FUNCTION_BLOCK TM_DI32 (* Composite Function Block Type *)
  (* Standard: 61499-2 *)
  (* Version 0.0, 18/08/2026, template *)
  PACKAGE Hidryco.HidrycoLib;
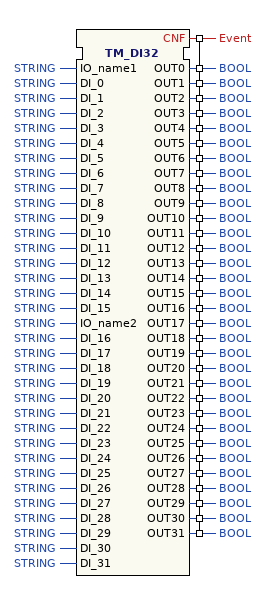
  EVENT_OUTPUT
    CNF WITH OUT0, OUT1, OUT2, OUT3, OUT4, OUT5, OUT6, OUT7, OUT8, OUT9, OUT10, OUT11, OUT12, OUT13, OUT14, OUT15, OUT16, OUT17, OUT18, OUT19, OUT20, OUT21, OUT22, OUT23, OUT24, OUT25, OUT26, OUT27, OUT28, OUT29, OUT30, OUT31;
  END_EVENT
  VAR_INPUT
    IO_name1 : STRING;
    DI_0 : STRING;
    DI_1 : STRING;
    DI_2 : STRING;
    DI_3 : STRING;
    DI_4 : STRING;
    DI_5 : STRING;
    DI_6 : STRING;
    DI_7 : STRING;
    DI_8 : STRING;
    DI_9 : STRING;
    DI_10 : STRING;
    DI_11 : STRING;
    DI_12 : STRING;
    DI_13 : STRING;
    DI_14 : STRING;
    DI_15 : STRING;
    IO_name2 : STRING;
    DI_16 : STRING;
    DI_17 : STRING;
    DI_18 : STRING;
    DI_19 : STRING;
    DI_20 : STRING;
    DI_21 : STRING;
    DI_22 : STRING;
    DI_23 : STRING;
    DI_24 : STRING;
    DI_25 : STRING;
    DI_26 : STRING;
    DI_27 : STRING;
    DI_28 : STRING;
    DI_29 : STRING;
    DI_30 : STRING;
    DI_31 : STRING;
  END_VAR
  VAR_OUTPUT
    OUT0 : BOOL; (* Output bit image, bit 0 is the LSB of OUT1 *)
    OUT1 : BOOL; (* Output bit image, bit 0 is the LSB of OUT1 *)
    OUT2 : BOOL; (* Output bit image, bit 0 is the LSB of OUT1 *)
    OUT3 : BOOL; (* Output bit image, bit 0 is the LSB of OUT1 *)
    OUT4 : BOOL; (* Output bit image, bit 0 is the LSB of OUT1 *)
    OUT5 : BOOL; (* Output bit image, bit 0 is the LSB of OUT1 *)
    OUT6 : BOOL; (* Output bit image, bit 0 is the LSB of OUT1 *)
    OUT7 : BOOL; (* Output bit image, bit 0 is the LSB of OUT1 *)
    OUT8 : BOOL; (* Output bit image, bit 0 is the LSB of OUT1 *)
    OUT9 : BOOL; (* Output bit image, bit 0 is the LSB of OUT1 *)
    OUT10 : BOOL; (* Output bit image, bit 0 is the LSB of OUT1 *)
    OUT11 : BOOL; (* Output bit image, bit 0 is the LSB of OUT1 *)
    OUT12 : BOOL; (* Output bit image, bit 0 is the LSB of OUT1 *)
    OUT13 : BOOL; (* Output bit image, bit 0 is the LSB of OUT1 *)
    OUT14 : BOOL; (* Output bit image, bit 0 is the LSB of OUT1 *)
    OUT15 : BOOL; (* Output bit image, bit 0 is the LSB of OUT1 *)
    OUT16 : BOOL; (* Output bit image, bit 0 is the LSB of OUT1 *)
    OUT17 : BOOL; (* Output bit image, bit 0 is the LSB of OUT1 *)
    OUT18 : BOOL; (* Output bit image, bit 0 is the LSB of OUT1 *)
    OUT19 : BOOL; (* Output bit image, bit 0 is the LSB of OUT1 *)
    OUT20 : BOOL; (* Output bit image, bit 0 is the LSB of OUT1 *)
    OUT21 : BOOL; (* Output bit image, bit 0 is the LSB of OUT1 *)
    OUT22 : BOOL; (* Output bit image, bit 0 is the LSB of OUT1 *)
    OUT23 : BOOL; (* Output bit image, bit 0 is the LSB of OUT1 *)
    OUT24 : BOOL; (* Output bit image, bit 0 is the LSB of OUT1 *)
    OUT25 : BOOL; (* Output bit image, bit 0 is the LSB of OUT1 *)
    OUT26 : BOOL; (* Output bit image, bit 0 is the LSB of OUT1 *)
    OUT27 : BOOL; (* Output bit image, bit 0 is the LSB of OUT1 *)
    OUT28 : BOOL; (* Output bit image, bit 0 is the LSB of OUT1 *)
    OUT29 : BOOL; (* Output bit image, bit 0 is the LSB of OUT1 *)
    OUT30 : BOOL; (* Output bit image, bit 0 is the LSB of OUT1 *)
    OUT31 : BOOL; (* Output bit image, bit 0 is the LSB of OUT1 *)
  END_VAR
  FBS
    BITMAN1 : BITMAN_1879143E4E6E9A030; {SET_ATTRIBUTE(Configuration.GenericFBType.InterfaceParams, Runtime.Standard#CNTIN:=1;CNTOUT:=16;IN${CNTIN$}:WORD;OUT${CNTOUT$}:BOOL,BOOL,BOOL,BOOL,BOOL,BOOL,BOOL,BOOL,BOOL,BOOL,BOOL,BOOL,BOOL,BOOL,BOOL,BOOL)}
    SYMLINKMULTIVARDST3 : SYMLINKMULTIVARDST_5A03F112CD5D470(QI := TRUE); {SET_ATTRIBUTE(Configuration.GenericFBType.InterfaceParams, Runtime.System#I:=1;VALUE${I$}:INT)}
    ANY2ANY1 : ANY2ANY_100577755E31233DE; {SET_ATTRIBUTE(Configuration.GenericFBType.InterfaceParams, Runtime.Standard#CNT:=1;IN${CNT$}:INT;OUT${CNT$}:WORD)}
    TM : SYMLINKMULTIVARSRC_854A896E88500D19(QI := TRUE); {SET_ATTRIBUTE(Configuration.GenericFBType.InterfaceParams, Runtime.System#I:=16;VALUE${I$}:BOOL,BOOL,BOOL,BOOL,BOOL,BOOL,BOOL,BOOL,BOOL,BOOL,BOOL,BOOL,BOOL,BOOL,BOOL,BOOL)}
    plcStart1 : plcStart(Prio := 3);
    BITMAN2 : BITMAN_1879143E4E6E9A030; {SET_ATTRIBUTE(Configuration.GenericFBType.InterfaceParams, Runtime.Standard#CNTIN:=1;CNTOUT:=16;IN${CNTIN$}:WORD;OUT${CNTOUT$}:BOOL,BOOL,BOOL,BOOL,BOOL,BOOL,BOOL,BOOL,BOOL,BOOL,BOOL,BOOL,BOOL,BOOL,BOOL,BOOL)}
    SYMLINKMULTIVARDST4 : SYMLINKMULTIVARDST_5A03F112CD5D470(QI := TRUE); {SET_ATTRIBUTE(Configuration.GenericFBType.InterfaceParams, Runtime.System#I:=1;VALUE${I$}:INT)}
    ANY2ANY2 : ANY2ANY_100577755E31233DE; {SET_ATTRIBUTE(Configuration.GenericFBType.InterfaceParams, Runtime.Standard#CNT:=1;IN${CNT$}:INT;OUT${CNT$}:WORD)}
    TM1 : SYMLINKMULTIVARSRC_854A896E88500D19(QI := TRUE); {SET_ATTRIBUTE(Configuration.GenericFBType.InterfaceParams, Runtime.System#I:=16;VALUE${I$}:BOOL,BOOL,BOOL,BOOL,BOOL,BOOL,BOOL,BOOL,BOOL,BOOL,BOOL,BOOL,BOOL,BOOL,BOOL,BOOL)}
    plcStart2 : plcStart(Prio := 3);
    FB1 : E_MERGE;
  END_FBS
  EVENT_CONNECTIONS
    SYMLINKMULTIVARDST3.CNF TO ANY2ANY1.REQ;
    ANY2ANY1.CNF TO BITMAN1.REQ;
    SYMLINKMULTIVARDST3.INITO TO BITMAN1.INIT;
    BITMAN1.INITO TO TM.INIT;
    BITMAN1.CNF TO TM.REQ;
    plcStart1.FIRST_INIT TO SYMLINKMULTIVARDST3.INIT;
    plcStart1.REDO_INIT TO SYMLINKMULTIVARDST3.INIT;
    TM.INITO TO plcStart1.ACK_FIRST;
    SYMLINKMULTIVARDST4.CNF TO ANY2ANY2.REQ;
    ANY2ANY2.CNF TO BITMAN2.REQ;
    SYMLINKMULTIVARDST4.INITO TO BITMAN2.INIT;
    BITMAN2.INITO TO TM1.INIT;
    BITMAN2.CNF TO TM1.REQ;
    plcStart2.FIRST_INIT TO SYMLINKMULTIVARDST4.INIT;
    plcStart2.REDO_INIT TO SYMLINKMULTIVARDST4.INIT;
    TM1.INITO TO plcStart2.ACK_FIRST;
    BITMAN2.CNF TO FB1.EI2;
    BITMAN1.CNF TO FB1.EI1;
    FB1.EO TO CNF;
  END_CONNECTIONS
  DATA_CONNECTIONS
    SYMLINKMULTIVARDST3.VALUE1 TO ANY2ANY1.IN1;
    ANY2ANY1.OUT1 TO BITMAN1.IN1;
    BITMAN1.OUT1 TO TM.VALUE1;
    BITMAN1.OUT2 TO TM.VALUE2;
    BITMAN1.OUT3 TO TM.VALUE3;
    BITMAN1.OUT4 TO TM.VALUE4;
    BITMAN1.OUT5 TO TM.VALUE5;
    BITMAN1.OUT6 TO TM.VALUE6;
    BITMAN1.OUT7 TO TM.VALUE7;
    BITMAN1.OUT8 TO TM.VALUE8;
    BITMAN1.OUT9 TO TM.VALUE9;
    BITMAN1.OUT10 TO TM.VALUE10;
    BITMAN1.OUT11 TO TM.VALUE11;
    BITMAN1.OUT12 TO TM.VALUE12;
    BITMAN1.OUT13 TO TM.VALUE13;
    BITMAN1.OUT14 TO TM.VALUE14;
    BITMAN1.OUT15 TO TM.VALUE15;
    BITMAN1.OUT16 TO TM.VALUE16;
    IO_name1 TO SYMLINKMULTIVARDST3.NAME1;
    DI_0 TO TM.NAME1;
    DI_1 TO TM.NAME2;
    DI_2 TO TM.NAME3;
    DI_3 TO TM.NAME4;
    DI_4 TO TM.NAME5;
    DI_5 TO TM.NAME6;
    DI_6 TO TM.NAME7;
    DI_7 TO TM.NAME8;
    DI_8 TO TM.NAME9;
    DI_9 TO TM.NAME10;
    DI_10 TO TM.NAME11;
    DI_11 TO TM.NAME12;
    DI_12 TO TM.NAME13;
    DI_13 TO TM.NAME14;
    DI_14 TO TM.NAME15;
    DI_15 TO TM.NAME16;
    SYMLINKMULTIVARDST4.VALUE1 TO ANY2ANY2.IN1;
    ANY2ANY2.OUT1 TO BITMAN2.IN1;
    BITMAN2.OUT1 TO TM1.VALUE1;
    BITMAN2.OUT2 TO TM1.VALUE2;
    BITMAN2.OUT3 TO TM1.VALUE3;
    BITMAN2.OUT4 TO TM1.VALUE4;
    BITMAN2.OUT5 TO TM1.VALUE5;
    BITMAN2.OUT6 TO TM1.VALUE6;
    BITMAN2.OUT7 TO TM1.VALUE7;
    BITMAN2.OUT8 TO TM1.VALUE8;
    BITMAN2.OUT9 TO TM1.VALUE9;
    BITMAN2.OUT10 TO TM1.VALUE10;
    BITMAN2.OUT11 TO TM1.VALUE11;
    BITMAN2.OUT12 TO TM1.VALUE12;
    BITMAN2.OUT13 TO TM1.VALUE13;
    BITMAN2.OUT14 TO TM1.VALUE14;
    BITMAN2.OUT15 TO TM1.VALUE15;
    BITMAN2.OUT16 TO TM1.VALUE16;
    IO_name2 TO SYMLINKMULTIVARDST4.NAME1;
    DI_16 TO TM1.NAME1;
    DI_17 TO TM1.NAME2;
    DI_18 TO TM1.NAME3;
    DI_19 TO TM1.NAME4;
    DI_20 TO TM1.NAME5;
    DI_21 TO TM1.NAME6;
    DI_22 TO TM1.NAME7;
    DI_23 TO TM1.NAME8;
    DI_24 TO TM1.NAME9;
    DI_25 TO TM1.NAME10;
    DI_26 TO TM1.NAME11;
    DI_27 TO TM1.NAME12;
    DI_28 TO TM1.NAME13;
    DI_29 TO TM1.NAME14;
    DI_30 TO TM1.NAME15;
    DI_31 TO TM1.NAME16;
    BITMAN1.OUT1 TO OUT0;
    BITMAN1.OUT2 TO OUT1;
    BITMAN1.OUT3 TO OUT2;
    BITMAN1.OUT4 TO OUT3;
    BITMAN1.OUT5 TO OUT4;
    BITMAN1.OUT6 TO OUT5;
    BITMAN1.OUT7 TO OUT6;
    BITMAN1.OUT8 TO OUT7;
    BITMAN1.OUT9 TO OUT8;
    BITMAN1.OUT10 TO OUT9;
    BITMAN1.OUT11 TO OUT10;
    BITMAN1.OUT12 TO OUT11;
    BITMAN1.OUT13 TO OUT12;
    BITMAN1.OUT14 TO OUT13;
    BITMAN1.OUT15 TO OUT14;
    BITMAN1.OUT16 TO OUT15;
    BITMAN2.OUT1 TO OUT16;
    BITMAN2.OUT2 TO OUT17;
    BITMAN2.OUT3 TO OUT18;
    BITMAN2.OUT4 TO OUT19;
    BITMAN2.OUT5 TO OUT20;
    BITMAN2.OUT6 TO OUT21;
    BITMAN2.OUT7 TO OUT22;
    BITMAN2.OUT8 TO OUT23;
    BITMAN2.OUT9 TO OUT24;
    BITMAN2.OUT10 TO OUT25;
    BITMAN2.OUT11 TO OUT26;
    BITMAN2.OUT12 TO OUT27;
    BITMAN2.OUT13 TO OUT28;
    BITMAN2.OUT14 TO OUT29;
    BITMAN2.OUT15 TO OUT30;
    BITMAN2.OUT16 TO OUT31;
  END_CONNECTIONS
END_FUNCTION_BLOCK
